INTERFACE I_Syntax_AdvancedDevice EXTENDS I_Syntax_BaseDevice

METHOD M_Configure : BOOL
VAR_INPUT
    stConfig : ST_Syntax_ComplexTree;
END_VAR
END_METHOD

METHOD M_GetDiagnostics : STRING(255)
VAR_OUTPUT
    nErrorCode : DINT;
END_VAR
END_METHOD

END_INTERFACE

(* stored: Version 1.1.0.1, ProductVersion 3.1.4024.16
   Itf I_Syntax_AdvancedDevice: Id {bb81855f-e08e-4c54-bae4-a3ed4fc19652}
   Method M_Configure: Id {e89cb159-6076-40ea-bc53-12a853453ef4}
   Method M_GetDiagnostics: Id {bc88c238-0bad-415b-9832-18420694ed9e} *)
